// TIA Portal V20 export
FUNCTION "06 T4 LANT Output" : Void   // FC1612, LAD
TITLE = OUTPUT
{ S7_Optimized_Access := 'TRUE' }
// stored: AutoNumber false, SetENOAutomatically false
   VAR_TEMP
      Aux_real : Real;
      Aux_dint : DInt;
      Aux_uint : UInt;
      Aux_Bool : Bool;
      Aux_OS : Bool;
   END_VAR
   VAR_TEMP   // added for the SCL form of the ladder/FBD networks
      _w1 : Bool;
      _w2 : Bool;
      _w3 : Bool;
   END_VAR
BEGIN

REGION Network 1: ============= INTERLOCKS MOVING FORWARD LANT =============
END_REGION

REGION Network 2: Interlocks Move FORWARD LANT - Permanent Conditions
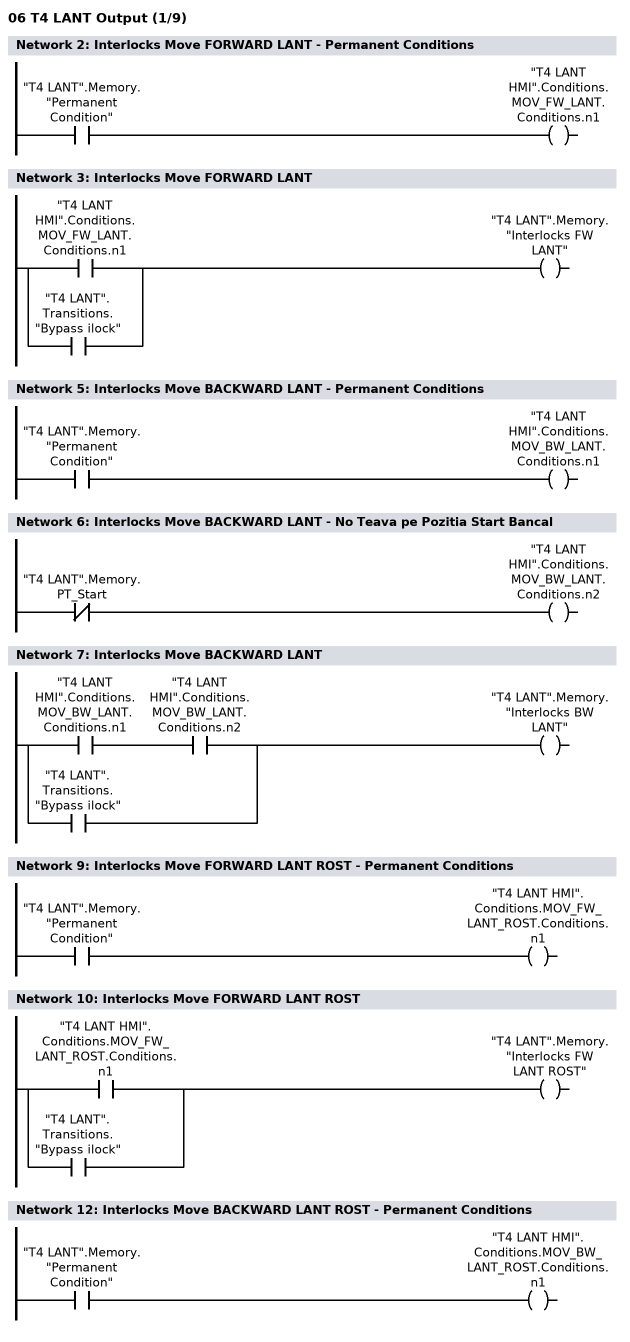
   RUNG wire#powerrail
      Contact( "T4 LANT".Memory."Permanent Condition" )
      Coil( "T4 LANT HMI".Conditions.MOV_FW_LANT.Conditions.n1 )
   END_RUNG
   // the same network as SCL:
   "T4 LANT HMI".Conditions.MOV_FW_LANT.Conditions.n1 := "T4 LANT".Memory."Permanent Condition";
END_REGION

REGION Network 3: Interlocks Move FORWARD LANT
   RUNG wire#powerrail
      Contact( "T4 LANT HMI".Conditions.MOV_FW_LANT.Conditions.n1 )
      wire#w1
      Coil( "T4 LANT".Memory."Interlocks FW LANT" )
   END_RUNG
   RUNG wire#powerrail
      Contact( "T4 LANT".Transitions."Bypass ilock" )
   END_RUNG wire#w1
   // the same network as SCL:
   "T4 LANT".Memory."Interlocks FW LANT" := "T4 LANT HMI".Conditions.MOV_FW_LANT.Conditions.n1 OR "T4 LANT".Transitions."Bypass ilock";
END_REGION

REGION Network 4: ============= INTERLOCKS MOVING BACKWARD LANT =============
END_REGION

REGION Network 5: Interlocks Move BACKWARD LANT - Permanent Conditions
   RUNG wire#powerrail
      Contact( "T4 LANT".Memory."Permanent Condition" )
      Coil( "T4 LANT HMI".Conditions.MOV_BW_LANT.Conditions.n1 )
   END_RUNG
   // the same network as SCL:
   "T4 LANT HMI".Conditions.MOV_BW_LANT.Conditions.n1 := "T4 LANT".Memory."Permanent Condition";
END_REGION

REGION Network 6: Interlocks Move BACKWARD LANT - No Teava pe Pozitia Start Bancal
   RUNG wire#powerrail
      I_Contact( "T4 LANT".Memory.PT_Start )
      Coil( "T4 LANT HMI".Conditions.MOV_BW_LANT.Conditions.n2 )
   END_RUNG
   // the same network as SCL:
   "T4 LANT HMI".Conditions.MOV_BW_LANT.Conditions.n2 := NOT "T4 LANT".Memory.PT_Start;
END_REGION

REGION Network 7: Interlocks Move BACKWARD LANT
   RUNG wire#powerrail
      Contact( "T4 LANT HMI".Conditions.MOV_BW_LANT.Conditions.n1 )
      Contact( "T4 LANT HMI".Conditions.MOV_BW_LANT.Conditions.n2 )
      wire#w1
      Coil( "T4 LANT".Memory."Interlocks BW LANT" )
   END_RUNG
   RUNG wire#powerrail
      Contact( "T4 LANT".Transitions."Bypass ilock" )
   END_RUNG wire#w1
   // the same network as SCL:
   "T4 LANT".Memory."Interlocks BW LANT" := ("T4 LANT HMI".Conditions.MOV_BW_LANT.Conditions.n1 AND "T4 LANT HMI".Conditions.MOV_BW_LANT.Conditions.n2) OR "T4 LANT".Transitions."Bypass ilock";
END_REGION

REGION Network 8: ============= INTERLOCKS MOVING FORWARD LANT ROST =============
END_REGION

REGION Network 9: Interlocks Move FORWARD LANT ROST - Permanent Conditions
   RUNG wire#powerrail
      Contact( "T4 LANT".Memory."Permanent Condition" )
      Coil( "T4 LANT HMI".Conditions.MOV_FW_LANT_ROST.Conditions.n1 )
   END_RUNG
   // the same network as SCL:
   "T4 LANT HMI".Conditions.MOV_FW_LANT_ROST.Conditions.n1 := "T4 LANT".Memory."Permanent Condition";
END_REGION

REGION Network 10: Interlocks Move FORWARD LANT ROST
   RUNG wire#powerrail
      Contact( "T4 LANT HMI".Conditions.MOV_FW_LANT_ROST.Conditions.n1 )
      wire#w1
      Coil( "T4 LANT".Memory."Interlocks FW LANT ROST" )
   END_RUNG
   RUNG wire#powerrail
      Contact( "T4 LANT".Transitions."Bypass ilock" )
   END_RUNG wire#w1
   // the same network as SCL:
   "T4 LANT".Memory."Interlocks FW LANT ROST" := "T4 LANT HMI".Conditions.MOV_FW_LANT_ROST.Conditions.n1 OR "T4 LANT".Transitions."Bypass ilock";
END_REGION

REGION Network 11: ============= INTERLOCKS MOVING BACKWARD LANT ROST =============
END_REGION

REGION Network 12: Interlocks Move BACKWARD LANT ROST - Permanent Conditions
   RUNG wire#powerrail
      Contact( "T4 LANT".Memory."Permanent Condition" )
      Coil( "T4 LANT HMI".Conditions.MOV_BW_LANT_ROST.Conditions.n1 )
   END_RUNG
   // the same network as SCL:
   "T4 LANT HMI".Conditions.MOV_BW_LANT_ROST.Conditions.n1 := "T4 LANT".Memory."Permanent Condition";
END_REGION

REGION Network 13: Interlocks Move BACKWARD LANT ROST - No TimeOut Cuplare/Decupl. Alim.Inv.LantRost
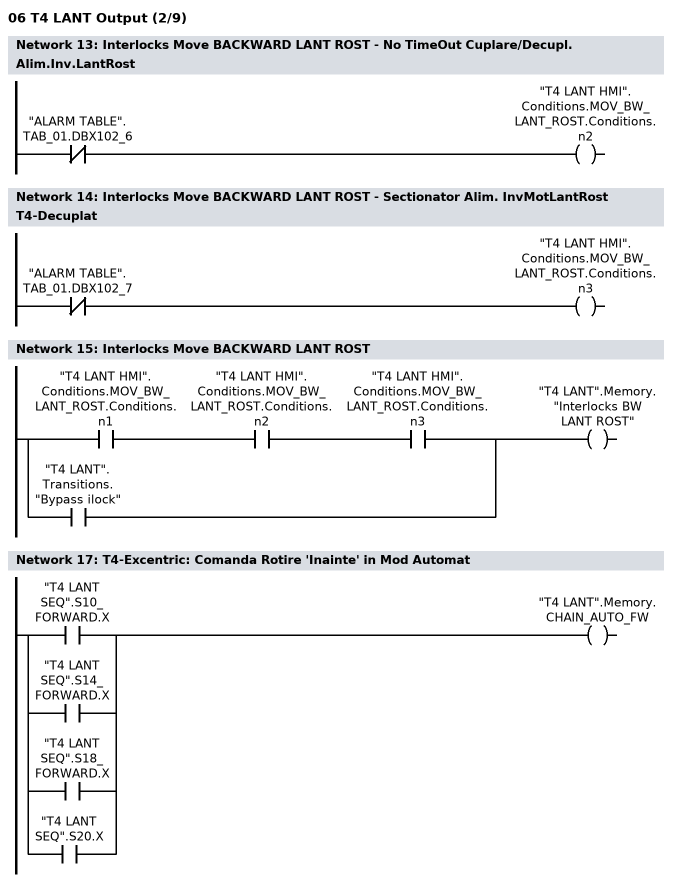
   RUNG wire#powerrail
      I_Contact( "ALARM TABLE".TAB_01.DBX102_6 )
      Coil( "T4 LANT HMI".Conditions.MOV_BW_LANT_ROST.Conditions.n2 )
   END_RUNG
   // the same network as SCL:
   "T4 LANT HMI".Conditions.MOV_BW_LANT_ROST.Conditions.n2 := NOT "ALARM TABLE".TAB_01.DBX102_6;
END_REGION

REGION Network 14: Interlocks Move BACKWARD LANT ROST - Sectionator Alim. InvMotLantRost T4-Decuplat
   RUNG wire#powerrail
      I_Contact( "ALARM TABLE".TAB_01.DBX102_7 )
      Coil( "T4 LANT HMI".Conditions.MOV_BW_LANT_ROST.Conditions.n3 )
   END_RUNG
   // the same network as SCL:
   "T4 LANT HMI".Conditions.MOV_BW_LANT_ROST.Conditions.n3 := NOT "ALARM TABLE".TAB_01.DBX102_7;
END_REGION

REGION Network 15: Interlocks Move BACKWARD LANT ROST
   RUNG wire#powerrail
      Contact( "T4 LANT HMI".Conditions.MOV_BW_LANT_ROST.Conditions.n1 )
      Contact( "T4 LANT HMI".Conditions.MOV_BW_LANT_ROST.Conditions.n2 )
      Contact( "T4 LANT HMI".Conditions.MOV_BW_LANT_ROST.Conditions.n3 )
      wire#w1
      Coil( "T4 LANT".Memory."Interlocks BW LANT ROST" )
   END_RUNG
   RUNG wire#powerrail
      Contact( "T4 LANT".Transitions."Bypass ilock" )
   END_RUNG wire#w1
   // the same network as SCL:
   "T4 LANT".Memory."Interlocks BW LANT ROST" := ("T4 LANT HMI".Conditions.MOV_BW_LANT_ROST.Conditions.n1 AND "T4 LANT HMI".Conditions.MOV_BW_LANT_ROST.Conditions.n2 AND "T4 LANT HMI".Conditions.MOV_BW_LANT_ROST.Conditions.n3) OR "T4 LANT".Transitions."Bypass ilock";
END_REGION

REGION Network 16: ============ COMMANDS ============
END_REGION

REGION Network 17: T4-Excentric: Comanda Rotire 'Inainte' in Mod Automat
   RUNG wire#powerrail
      Contact( "T4 LANT SEQ".S10_FORWARD.X )
      wire#w1
      Coil( "T4 LANT".Memory.CHAIN_AUTO_FW )
   END_RUNG
   RUNG wire#powerrail
      Contact( "T4 LANT SEQ".S14_FORWARD.X )
   END_RUNG wire#w1
   RUNG wire#powerrail
      Contact( "T4 LANT SEQ".S18_FORWARD.X )
   END_RUNG wire#w1
   RUNG wire#powerrail
      Contact( "T4 LANT SEQ".S20.X )
   END_RUNG wire#w1
   // the same network as SCL:
   "T4 LANT".Memory.CHAIN_AUTO_FW := "T4 LANT SEQ".S10_FORWARD.X OR "T4 LANT SEQ".S14_FORWARD.X OR "T4 LANT SEQ".S18_FORWARD.X OR "T4 LANT SEQ".S20.X;
END_REGION

REGION Network 18: T4-Lant: Deplasare 'Inainte'
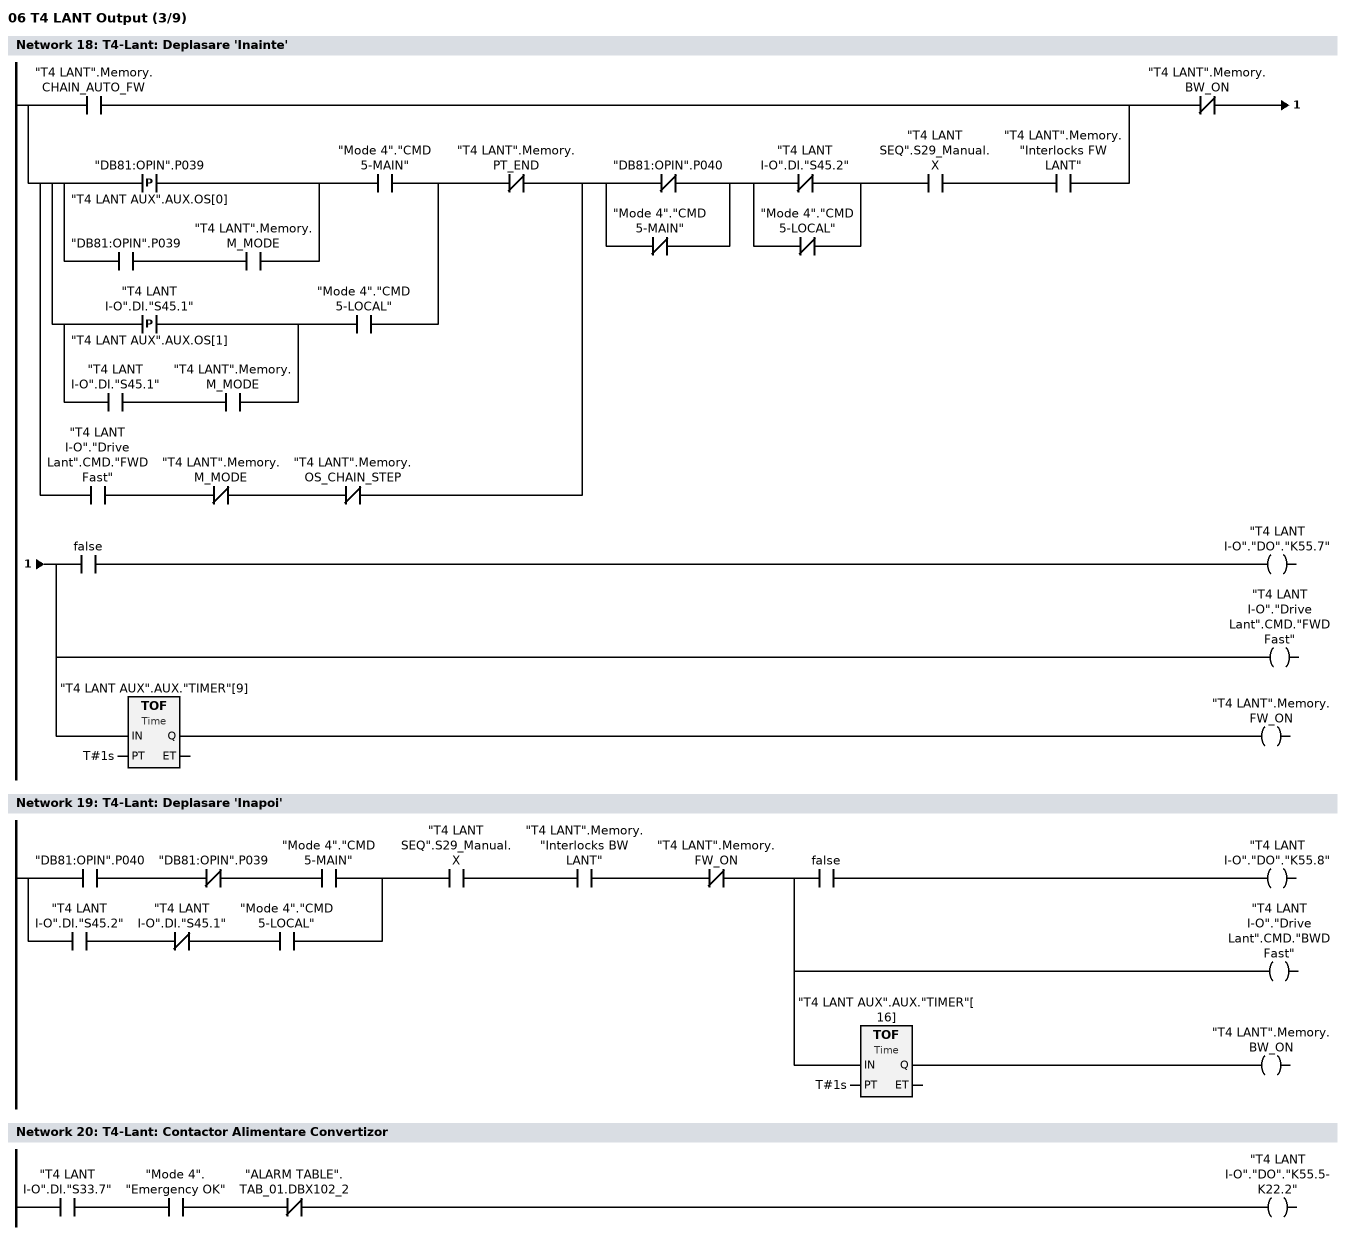
   RUNG wire#powerrail
      Contact( "T4 LANT".Memory.CHAIN_AUTO_FW )
      wire#w1
      I_Contact( "T4 LANT".Memory.BW_ON )
      wire#w8
      Contact( false )
      Coil( "T4 LANT I-O"."DO"."K55.7" )
   END_RUNG
   RUNG wire#powerrail
      P_Contact(operand := "DB81:OPIN".P039, bit := "T4 LANT AUX".AUX.OS[0])
      wire#w2
      Contact( "Mode 4"."CMD 5-MAIN" )
      wire#w3
      I_Contact( "T4 LANT".Memory.PT_END )
      wire#w5
      I_Contact( "DB81:OPIN".P040 )
      wire#w6
      I_Contact( "T4 LANT I-O".DI."S45.2" )
      wire#w7
      Contact( "T4 LANT SEQ".S29_Manual.X )
      Contact( "T4 LANT".Memory."Interlocks FW LANT" )
   END_RUNG wire#w1
   RUNG wire#powerrail
      Contact( "DB81:OPIN".P039 )
      Contact( "T4 LANT".Memory.M_MODE )
   END_RUNG wire#w2
   RUNG wire#powerrail
      P_Contact(operand := "T4 LANT I-O".DI."S45.1", bit := "T4 LANT AUX".AUX.OS[1])
      wire#w4
      Contact( "Mode 4"."CMD 5-LOCAL" )
   END_RUNG wire#w3
   RUNG wire#powerrail
      Contact( "T4 LANT I-O".DI."S45.1" )
      Contact( "T4 LANT".Memory.M_MODE )
   END_RUNG wire#w4
   RUNG wire#powerrail
      Contact( "T4 LANT I-O"."Drive Lant".CMD."FWD Fast" )
      I_Contact( "T4 LANT".Memory.M_MODE )
      I_Contact( "T4 LANT".Memory.OS_CHAIN_STEP )
   END_RUNG wire#w5
   RUNG wire#w5
      I_Contact( "Mode 4"."CMD 5-MAIN" )
   END_RUNG wire#w6
   RUNG wire#w6
      I_Contact( "Mode 4"."CMD 5-LOCAL" )
   END_RUNG wire#w7
   RUNG wire#w8
      Coil( "T4 LANT I-O"."Drive Lant".CMD."FWD Fast" )
   END_RUNG
   RUNG wire#w8
      { S7_Templates := "time_type := Time" } "T4 LANT AUX".AUX."TIMER"[9].TOF(pt := T#1s, et =>)
      Coil( "T4 LANT".Memory.FW_ON )
   END_RUNG
   // the same network as SCL:
   #_w1 := "DB81:OPIN".P039 AND NOT "T4 LANT AUX".AUX.OS[0];   // rising edge of "DB81:OPIN".P039
   "T4 LANT AUX".AUX.OS[0] := "DB81:OPIN".P039;
   #_w2 := "T4 LANT I-O".DI."S45.1" AND NOT "T4 LANT AUX".AUX.OS[1];   // rising edge of "T4 LANT I-O".DI."S45.1"
   "T4 LANT AUX".AUX.OS[1] := "T4 LANT I-O".DI."S45.1";
   #_w3 := ("T4 LANT".Memory.CHAIN_AUTO_FW OR ((((((#_w1 OR ("DB81:OPIN".P039 AND "T4 LANT".Memory.M_MODE)) AND "Mode 4"."CMD 5-MAIN") OR ((#_w2 OR ("T4 LANT I-O".DI."S45.1" AND "T4 LANT".Memory.M_MODE)) AND "Mode 4"."CMD 5-LOCAL")) AND NOT "T4 LANT".Memory.PT_END) OR ("T4 LANT I-O"."Drive Lant".CMD."FWD Fast" AND NOT "T4 LANT".Memory.M_MODE AND NOT "T4 LANT".Memory.OS_CHAIN_STEP)) AND (NOT "DB81:OPIN".P040 OR NOT "Mode 4"."CMD 5-MAIN") AND (NOT "T4 LANT I-O".DI."S45.2" OR NOT "Mode 4"."CMD 5-LOCAL") AND "T4 LANT SEQ".S29_Manual.X AND "T4 LANT".Memory."Interlocks FW LANT")) AND NOT "T4 LANT".Memory.BW_ON;
   "T4 LANT I-O"."DO"."K55.7" := #_w3 AND false;
   "T4 LANT I-O"."Drive Lant".CMD."FWD Fast" := #_w3;
   "T4 LANT AUX".AUX."TIMER"[9].TOF(IN := #_w3, PT := T#1s);
   "T4 LANT".Memory.FW_ON := "T4 LANT AUX".AUX."TIMER"[9].Q;
END_REGION

REGION Network 19: T4-Lant: Deplasare 'Inapoi'
   RUNG wire#powerrail
      Contact( "DB81:OPIN".P040 )
      I_Contact( "DB81:OPIN".P039 )
      Contact( "Mode 4"."CMD 5-MAIN" )
      wire#w1
      Contact( "T4 LANT SEQ".S29_Manual.X )
      Contact( "T4 LANT".Memory."Interlocks BW LANT" )
      I_Contact( "T4 LANT".Memory.FW_ON )
      wire#w2
      Contact( false )
      Coil( "T4 LANT I-O"."DO"."K55.8" )
   END_RUNG
   RUNG wire#powerrail
      Contact( "T4 LANT I-O".DI."S45.2" )
      I_Contact( "T4 LANT I-O".DI."S45.1" )
      Contact( "Mode 4"."CMD 5-LOCAL" )
   END_RUNG wire#w1
   RUNG wire#w2
      Coil( "T4 LANT I-O"."Drive Lant".CMD."BWD Fast" )
   END_RUNG
   RUNG wire#w2
      { S7_Templates := "time_type := Time" } "T4 LANT AUX".AUX."TIMER"[16].TOF(pt := T#1s, et =>)
      Coil( "T4 LANT".Memory.BW_ON )
   END_RUNG
   // the same network as SCL:
   #_w1 := (("DB81:OPIN".P040 AND NOT "DB81:OPIN".P039 AND "Mode 4"."CMD 5-MAIN") OR ("T4 LANT I-O".DI."S45.2" AND NOT "T4 LANT I-O".DI."S45.1" AND "Mode 4"."CMD 5-LOCAL")) AND "T4 LANT SEQ".S29_Manual.X AND "T4 LANT".Memory."Interlocks BW LANT" AND NOT "T4 LANT".Memory.FW_ON;
   "T4 LANT I-O"."DO"."K55.8" := #_w1 AND false;
   "T4 LANT I-O"."Drive Lant".CMD."BWD Fast" := #_w1;
   "T4 LANT AUX".AUX."TIMER"[16].TOF(IN := #_w1, PT := T#1s);
   "T4 LANT".Memory.BW_ON := "T4 LANT AUX".AUX."TIMER"[16].Q;
END_REGION

REGION Network 20: T4-Lant: Contactor Alimentare Convertizor
   RUNG wire#powerrail
      Contact( "T4 LANT I-O".DI."S33.7" )
      Contact( "Mode 4"."Emergency OK" )
      I_Contact( "ALARM TABLE".TAB_01.DBX102_2 )
      Coil( "T4 LANT I-O"."DO"."K55.5-K22.2" )
   END_RUNG
   // the same network as SCL:
   "T4 LANT I-O"."DO"."K55.5-K22.2" := "T4 LANT I-O".DI."S33.7" AND "Mode 4"."Emergency OK" AND NOT "ALARM TABLE".TAB_01.DBX102_2;
END_REGION

REGION Network 21: T4-LantRost: Comanda Deplasare 'Inainte'
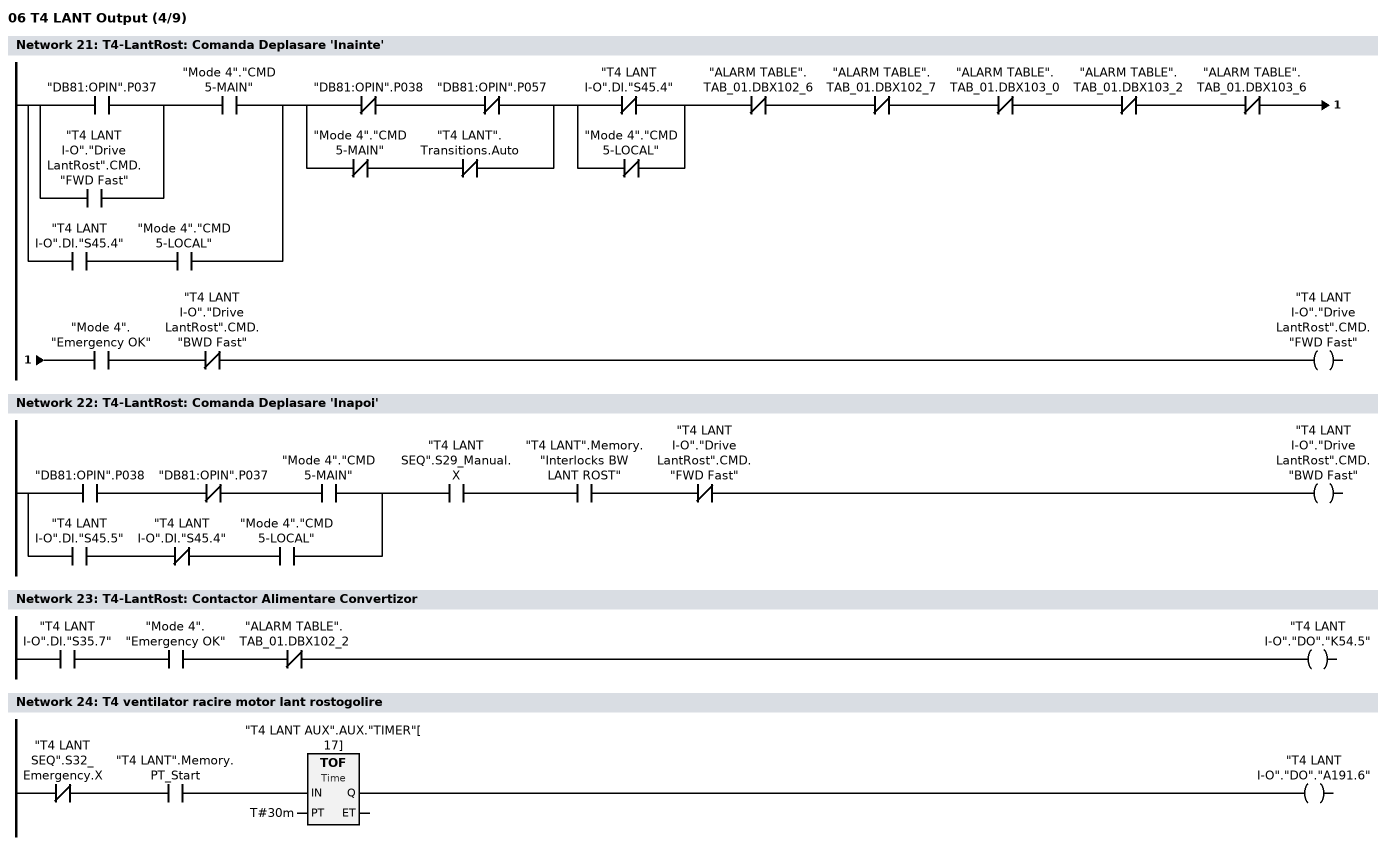
   RUNG wire#powerrail
      Contact( "DB81:OPIN".P037 )
      wire#w1
      Contact( "Mode 4"."CMD 5-MAIN" )
      wire#w2
      I_Contact( "DB81:OPIN".P038 )
      I_Contact( "DB81:OPIN".P057 )
      wire#w3
      I_Contact( "T4 LANT I-O".DI."S45.4" )
      wire#w4
      I_Contact( "ALARM TABLE".TAB_01.DBX102_6 )
      I_Contact( "ALARM TABLE".TAB_01.DBX102_7 )
      I_Contact( "ALARM TABLE".TAB_01.DBX103_0 )
      I_Contact( "ALARM TABLE".TAB_01.DBX103_2 )
      I_Contact( "ALARM TABLE".TAB_01.DBX103_6 )
      Contact( "Mode 4"."Emergency OK" )
      I_Contact( "T4 LANT I-O"."Drive LantRost".CMD."BWD Fast" )
      Coil( "T4 LANT I-O"."Drive LantRost".CMD."FWD Fast" )
   END_RUNG
   RUNG wire#powerrail
      Contact( "T4 LANT I-O"."Drive LantRost".CMD."FWD Fast" )
   END_RUNG wire#w1
   RUNG wire#powerrail
      Contact( "T4 LANT I-O".DI."S45.4" )
      Contact( "Mode 4"."CMD 5-LOCAL" )
   END_RUNG wire#w2
   RUNG wire#w2
      I_Contact( "Mode 4"."CMD 5-MAIN" )
      I_Contact( "T4 LANT".Transitions.Auto )
   END_RUNG wire#w3
   RUNG wire#w3
      I_Contact( "Mode 4"."CMD 5-LOCAL" )
   END_RUNG wire#w4
   // the same network as SCL:
   "T4 LANT I-O"."Drive LantRost".CMD."FWD Fast" := ((("DB81:OPIN".P037 OR "T4 LANT I-O"."Drive LantRost".CMD."FWD Fast") AND "Mode 4"."CMD 5-MAIN") OR ("T4 LANT I-O".DI."S45.4" AND "Mode 4"."CMD 5-LOCAL")) AND ((NOT "DB81:OPIN".P038 AND NOT "DB81:OPIN".P057) OR (NOT "Mode 4"."CMD 5-MAIN" AND NOT "T4 LANT".Transitions.Auto)) AND (NOT "T4 LANT I-O".DI."S45.4" OR NOT "Mode 4"."CMD 5-LOCAL") AND NOT "ALARM TABLE".TAB_01.DBX102_6 AND NOT "ALARM TABLE".TAB_01.DBX102_7 AND NOT "ALARM TABLE".TAB_01.DBX103_0 AND NOT "ALARM TABLE".TAB_01.DBX103_2 AND NOT "ALARM TABLE".TAB_01.DBX103_6 AND "Mode 4"."Emergency OK" AND NOT "T4 LANT I-O"."Drive LantRost".CMD."BWD Fast";
END_REGION

REGION Network 22: T4-LantRost: Comanda Deplasare 'Inapoi'
   RUNG wire#powerrail
      Contact( "DB81:OPIN".P038 )
      I_Contact( "DB81:OPIN".P037 )
      Contact( "Mode 4"."CMD 5-MAIN" )
      wire#w1
      Contact( "T4 LANT SEQ".S29_Manual.X )
      Contact( "T4 LANT".Memory."Interlocks BW LANT ROST" )
      I_Contact( "T4 LANT I-O"."Drive LantRost".CMD."FWD Fast" )
      Coil( "T4 LANT I-O"."Drive LantRost".CMD."BWD Fast" )
   END_RUNG
   RUNG wire#powerrail
      Contact( "T4 LANT I-O".DI."S45.5" )
      I_Contact( "T4 LANT I-O".DI."S45.4" )
      Contact( "Mode 4"."CMD 5-LOCAL" )
   END_RUNG wire#w1
   // the same network as SCL:
   "T4 LANT I-O"."Drive LantRost".CMD."BWD Fast" := (("DB81:OPIN".P038 AND NOT "DB81:OPIN".P037 AND "Mode 4"."CMD 5-MAIN") OR ("T4 LANT I-O".DI."S45.5" AND NOT "T4 LANT I-O".DI."S45.4" AND "Mode 4"."CMD 5-LOCAL")) AND "T4 LANT SEQ".S29_Manual.X AND "T4 LANT".Memory."Interlocks BW LANT ROST" AND NOT "T4 LANT I-O"."Drive LantRost".CMD."FWD Fast";
END_REGION

REGION Network 23: T4-LantRost: Contactor Alimentare Convertizor
   RUNG wire#powerrail
      Contact( "T4 LANT I-O".DI."S35.7" )
      Contact( "Mode 4"."Emergency OK" )
      I_Contact( "ALARM TABLE".TAB_01.DBX102_2 )
      Coil( "T4 LANT I-O"."DO"."K54.5" )
   END_RUNG
   // the same network as SCL:
   "T4 LANT I-O"."DO"."K54.5" := "T4 LANT I-O".DI."S35.7" AND "Mode 4"."Emergency OK" AND NOT "ALARM TABLE".TAB_01.DBX102_2;
END_REGION

REGION Network 24: T4 ventilator racire motor lant rostogolire
   RUNG wire#powerrail
      I_Contact( "T4 LANT SEQ".S32_Emergency.X )
      Contact( "T4 LANT".Memory.PT_Start )
      { S7_Templates := "time_type := Time" } "T4 LANT AUX".AUX."TIMER"[17].TOF(pt := T#30m, et =>)
      Coil( "T4 LANT I-O"."DO"."A191.6" )
   END_RUNG
   // the same network as SCL:
   "T4 LANT AUX".AUX."TIMER"[17].TOF(IN := NOT "T4 LANT SEQ".S32_Emergency.X AND "T4 LANT".Memory.PT_Start,
                           PT := T#30m);
   "T4 LANT I-O"."DO"."A191.6" := "T4 LANT AUX".AUX."TIMER"[17].Q;
END_REGION

REGION Network 25: T4-Lant: Ciclu Rapid: Viteza Referinta Incarcare
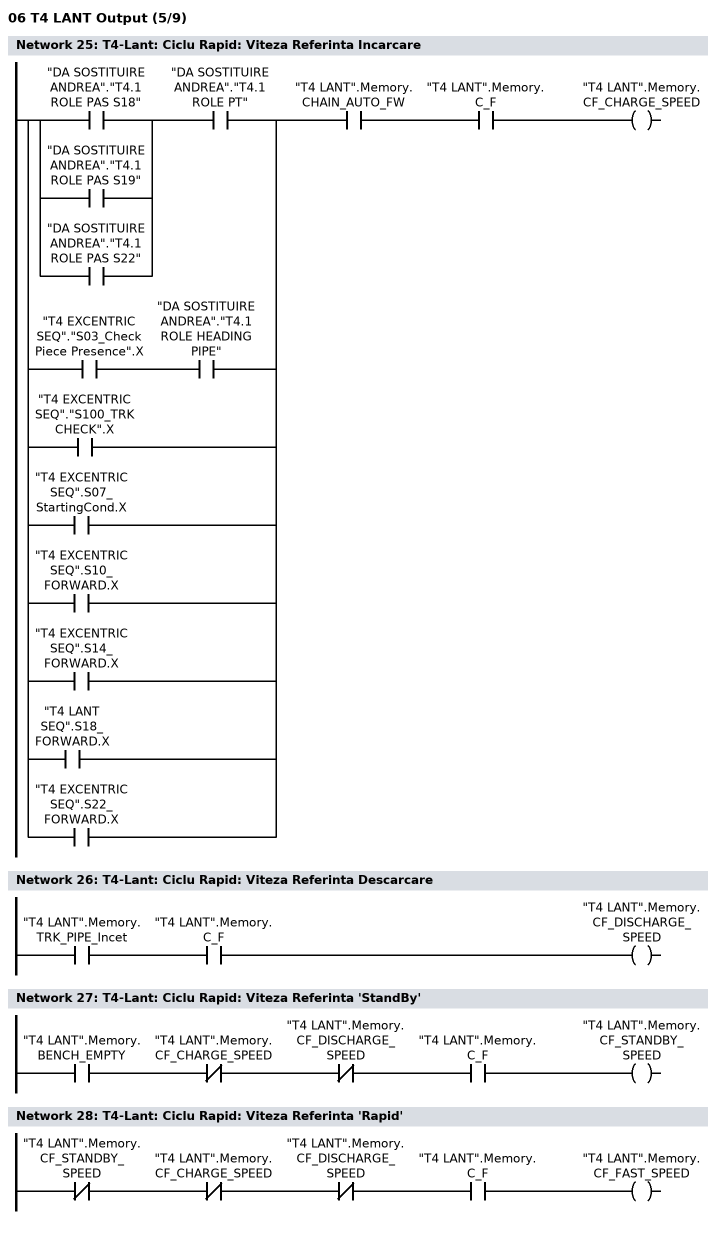
   RUNG wire#powerrail
      Contact( "DA SOSTITUIRE ANDREA"."T4.1 ROLE PAS S18" )
      wire#w1
      Contact( "DA SOSTITUIRE ANDREA"."T4.1 ROLE PT" )
      wire#w2
      Contact( "T4 LANT".Memory.CHAIN_AUTO_FW )
      Contact( "T4 LANT".Memory.C_F )
      Coil( "T4 LANT".Memory.CF_CHARGE_SPEED )
   END_RUNG
   RUNG wire#powerrail
      Contact( "DA SOSTITUIRE ANDREA"."T4.1 ROLE PAS S19" )
   END_RUNG wire#w1
   RUNG wire#powerrail
      Contact( "DA SOSTITUIRE ANDREA"."T4.1 ROLE PAS S22" )
   END_RUNG wire#w1
   RUNG wire#powerrail
      Contact( "T4 EXCENTRIC SEQ"."S03_Check Piece Presence".X )
      Contact( "DA SOSTITUIRE ANDREA"."T4.1 ROLE HEADING PIPE" )
   END_RUNG wire#w2
   RUNG wire#powerrail
      Contact( "T4 EXCENTRIC SEQ"."S100_TRK CHECK".X )
   END_RUNG wire#w2
   RUNG wire#powerrail
      Contact( "T4 EXCENTRIC SEQ".S07_StartingCond.X )
   END_RUNG wire#w2
   RUNG wire#powerrail
      Contact( "T4 EXCENTRIC SEQ".S10_FORWARD.X )
   END_RUNG wire#w2
   RUNG wire#powerrail
      Contact( "T4 EXCENTRIC SEQ".S14_FORWARD.X )
   END_RUNG wire#w2
   RUNG wire#powerrail
      Contact( "T4 LANT SEQ".S18_FORWARD.X )
   END_RUNG wire#w2
   RUNG wire#powerrail
      Contact( "T4 EXCENTRIC SEQ".S22_FORWARD.X )
   END_RUNG wire#w2
   // the same network as SCL:
   "T4 LANT".Memory.CF_CHARGE_SPEED := ((("DA SOSTITUIRE ANDREA"."T4.1 ROLE PAS S18" OR "DA SOSTITUIRE ANDREA"."T4.1 ROLE PAS S19" OR "DA SOSTITUIRE ANDREA"."T4.1 ROLE PAS S22") AND "DA SOSTITUIRE ANDREA"."T4.1 ROLE PT") OR ("T4 EXCENTRIC SEQ"."S03_Check Piece Presence".X AND "DA SOSTITUIRE ANDREA"."T4.1 ROLE HEADING PIPE") OR "T4 EXCENTRIC SEQ"."S100_TRK CHECK".X OR "T4 EXCENTRIC SEQ".S07_StartingCond.X OR "T4 EXCENTRIC SEQ".S10_FORWARD.X OR "T4 EXCENTRIC SEQ".S14_FORWARD.X OR "T4 LANT SEQ".S18_FORWARD.X OR "T4 EXCENTRIC SEQ".S22_FORWARD.X) AND "T4 LANT".Memory.CHAIN_AUTO_FW AND "T4 LANT".Memory.C_F;
END_REGION

REGION Network 26: T4-Lant: Ciclu Rapid: Viteza Referinta Descarcare
   RUNG wire#powerrail
      Contact( "T4 LANT".Memory.TRK_PIPE_Incet )
      Contact( "T4 LANT".Memory.C_F )
      Coil( "T4 LANT".Memory.CF_DISCHARGE_SPEED )
   END_RUNG
   // the same network as SCL:
   "T4 LANT".Memory.CF_DISCHARGE_SPEED := "T4 LANT".Memory.TRK_PIPE_Incet AND "T4 LANT".Memory.C_F;
END_REGION

REGION Network 27: T4-Lant: Ciclu Rapid: Viteza Referinta 'StandBy'
   RUNG wire#powerrail
      Contact( "T4 LANT".Memory.BENCH_EMPTY )
      I_Contact( "T4 LANT".Memory.CF_CHARGE_SPEED )
      I_Contact( "T4 LANT".Memory.CF_DISCHARGE_SPEED )
      Contact( "T4 LANT".Memory.C_F )
      Coil( "T4 LANT".Memory.CF_STANDBY_SPEED )
   END_RUNG
   // the same network as SCL:
   "T4 LANT".Memory.CF_STANDBY_SPEED := "T4 LANT".Memory.BENCH_EMPTY AND NOT "T4 LANT".Memory.CF_CHARGE_SPEED AND NOT "T4 LANT".Memory.CF_DISCHARGE_SPEED AND "T4 LANT".Memory.C_F;
END_REGION

REGION Network 28: T4-Lant: Ciclu Rapid: Viteza Referinta 'Rapid'
   RUNG wire#powerrail
      I_Contact( "T4 LANT".Memory.CF_STANDBY_SPEED )
      I_Contact( "T4 LANT".Memory.CF_CHARGE_SPEED )
      I_Contact( "T4 LANT".Memory.CF_DISCHARGE_SPEED )
      Contact( "T4 LANT".Memory.C_F )
      Coil( "T4 LANT".Memory.CF_FAST_SPEED )
   END_RUNG
   // the same network as SCL:
   "T4 LANT".Memory.CF_FAST_SPEED := NOT "T4 LANT".Memory.CF_STANDBY_SPEED AND NOT "T4 LANT".Memory.CF_CHARGE_SPEED AND NOT "T4 LANT".Memory.CF_DISCHARGE_SPEED AND "T4 LANT".Memory.C_F;
END_REGION

REGION Network 29: T4-Lant: Viteza Teava 'Inainte' in Mod Automat [m/min *10]
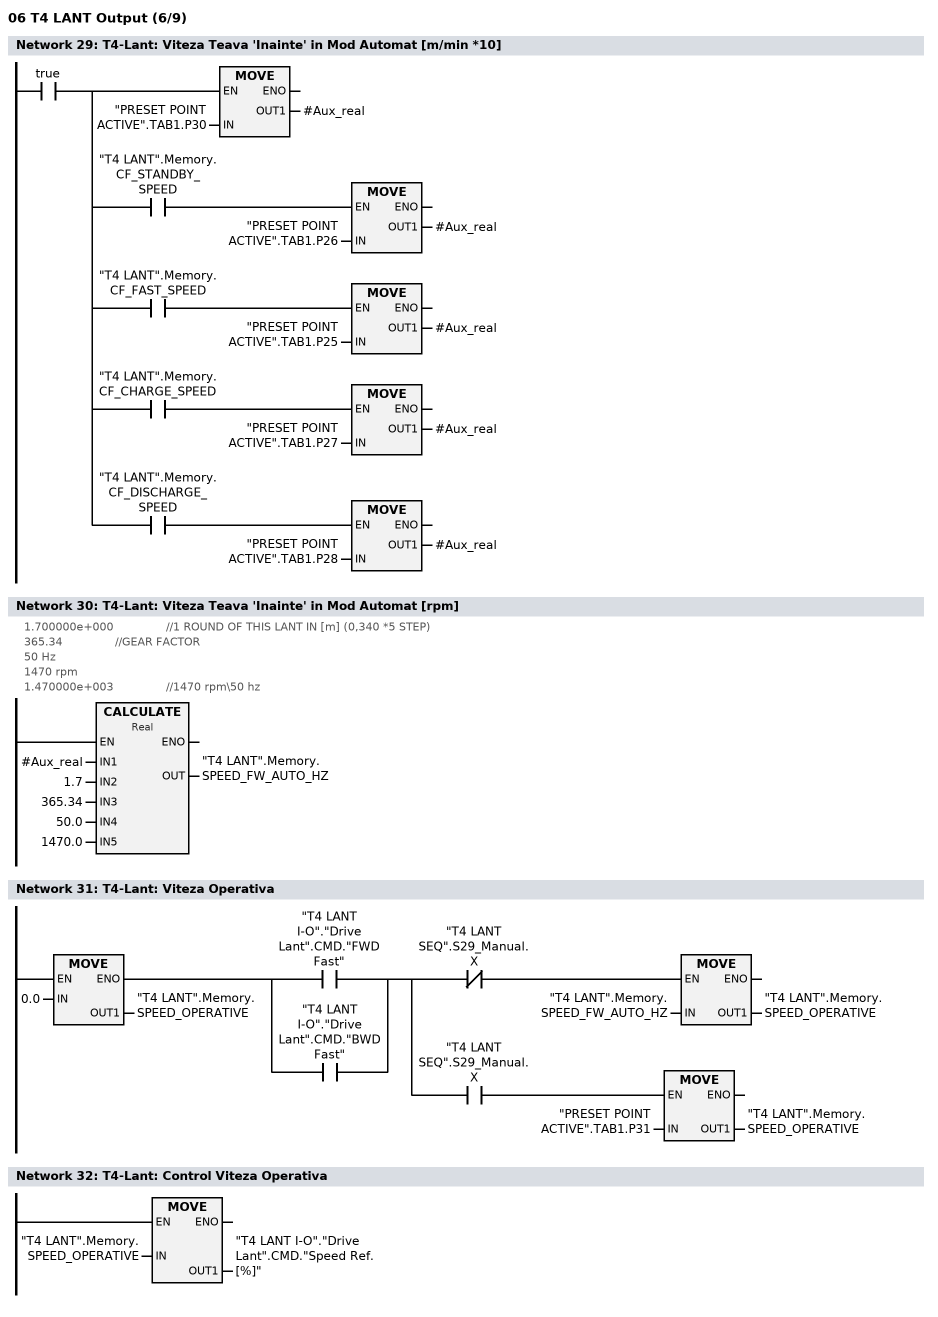
   RUNG wire#powerrail
      Contact( true )
      wire#w1
      Move(in := "PRESET POINT ACTIVE".TAB1.P30, out1 => #Aux_real)
   END_RUNG
   RUNG wire#w1
      Contact( "T4 LANT".Memory.CF_STANDBY_SPEED )
      Move(in := "PRESET POINT ACTIVE".TAB1.P26, out1 => #Aux_real)
   END_RUNG
   RUNG wire#w1
      Contact( "T4 LANT".Memory.CF_FAST_SPEED )
      Move(in := "PRESET POINT ACTIVE".TAB1.P25, out1 => #Aux_real)
   END_RUNG
   RUNG wire#w1
      Contact( "T4 LANT".Memory.CF_CHARGE_SPEED )
      Move(in := "PRESET POINT ACTIVE".TAB1.P27, out1 => #Aux_real)
   END_RUNG
   RUNG wire#w1
      Contact( "T4 LANT".Memory.CF_DISCHARGE_SPEED )
      Move(in := "PRESET POINT ACTIVE".TAB1.P28, out1 => #Aux_real)
   END_RUNG
   // the same network as SCL:
   IF true THEN #Aux_real := "PRESET POINT ACTIVE".TAB1.P30; END_IF;
   IF true AND "T4 LANT".Memory.CF_STANDBY_SPEED THEN #Aux_real := "PRESET POINT ACTIVE".TAB1.P26; END_IF;
   IF true AND "T4 LANT".Memory.CF_FAST_SPEED THEN #Aux_real := "PRESET POINT ACTIVE".TAB1.P25; END_IF;
   IF true AND "T4 LANT".Memory.CF_CHARGE_SPEED THEN #Aux_real := "PRESET POINT ACTIVE".TAB1.P27; END_IF;
   IF true AND "T4 LANT".Memory.CF_DISCHARGE_SPEED THEN #Aux_real := "PRESET POINT ACTIVE".TAB1.P28; END_IF;
END_REGION

REGION Network 30: T4-Lant: Viteza Teava 'Inainte' in Mod Automat [rpm]
   // 1.700000e+000               //1 ROUND OF THIS LANT IN [m] (0,340 *5 STEP) 
   //  365.34               //GEAR FACTOR
   // 50 Hz
   // 1470 rpm
   // 1.470000e+003               //1470 rpm\50 hz
   RUNG wire#powerrail
      { S7_Templates := "SrcType := Real"; S7_Expression := "IN1/IN2*IN3*IN4/IN5" } Calculate(in1 := #Aux_real, in2 := 1.7, in3 := 365.34, in4 := 50.0, in5 := 1470.0, out => "T4 LANT".Memory.SPEED_FW_AUTO_HZ)
   END_RUNG
   // the same network as SCL:
   "T4 LANT".Memory.SPEED_FW_AUTO_HZ := #Aux_real/1.7*365.34*50.0/1470.0;
END_REGION

REGION Network 31: T4-Lant: Viteza Operativa
   RUNG wire#powerrail
      Move(in := 0.0, out1 => "T4 LANT".Memory.SPEED_OPERATIVE)
      wire#w1
      Contact( "T4 LANT I-O"."Drive Lant".CMD."FWD Fast" )
      wire#w2
      I_Contact( "T4 LANT SEQ".S29_Manual.X )
      Move(in := "T4 LANT".Memory.SPEED_FW_AUTO_HZ, out1 => "T4 LANT".Memory.SPEED_OPERATIVE)
   END_RUNG
   RUNG wire#w1
      Contact( "T4 LANT I-O"."Drive Lant".CMD."BWD Fast" )
   END_RUNG wire#w2
   RUNG wire#w2
      Contact( "T4 LANT SEQ".S29_Manual.X )
      Move(in := "PRESET POINT ACTIVE".TAB1.P31, out1 => "T4 LANT".Memory.SPEED_OPERATIVE)
   END_RUNG
   // the same network as SCL:
   "T4 LANT".Memory.SPEED_OPERATIVE := 0.0;
   #_w1 := "T4 LANT I-O"."Drive Lant".CMD."FWD Fast" OR "T4 LANT I-O"."Drive Lant".CMD."BWD Fast";
   IF #_w1 AND NOT "T4 LANT SEQ".S29_Manual.X THEN
       "T4 LANT".Memory.SPEED_OPERATIVE := "T4 LANT".Memory.SPEED_FW_AUTO_HZ;
   END_IF;
   IF #_w1 AND "T4 LANT SEQ".S29_Manual.X THEN
       "T4 LANT".Memory.SPEED_OPERATIVE := "PRESET POINT ACTIVE".TAB1.P31;
   END_IF;
END_REGION

REGION Network 32: T4-Lant: Control Viteza Operativa
   RUNG wire#powerrail
      Move(in := "T4 LANT".Memory.SPEED_OPERATIVE, out1 => "T4 LANT I-O"."Drive Lant".CMD."Speed Ref. [%]")
   END_RUNG
   // the same network as SCL:
   "T4 LANT I-O"."Drive Lant".CMD."Speed Ref. [%]" := "T4 LANT".Memory.SPEED_OPERATIVE;
END_REGION

REGION Network 33: T4-Lant: Contactor Frana
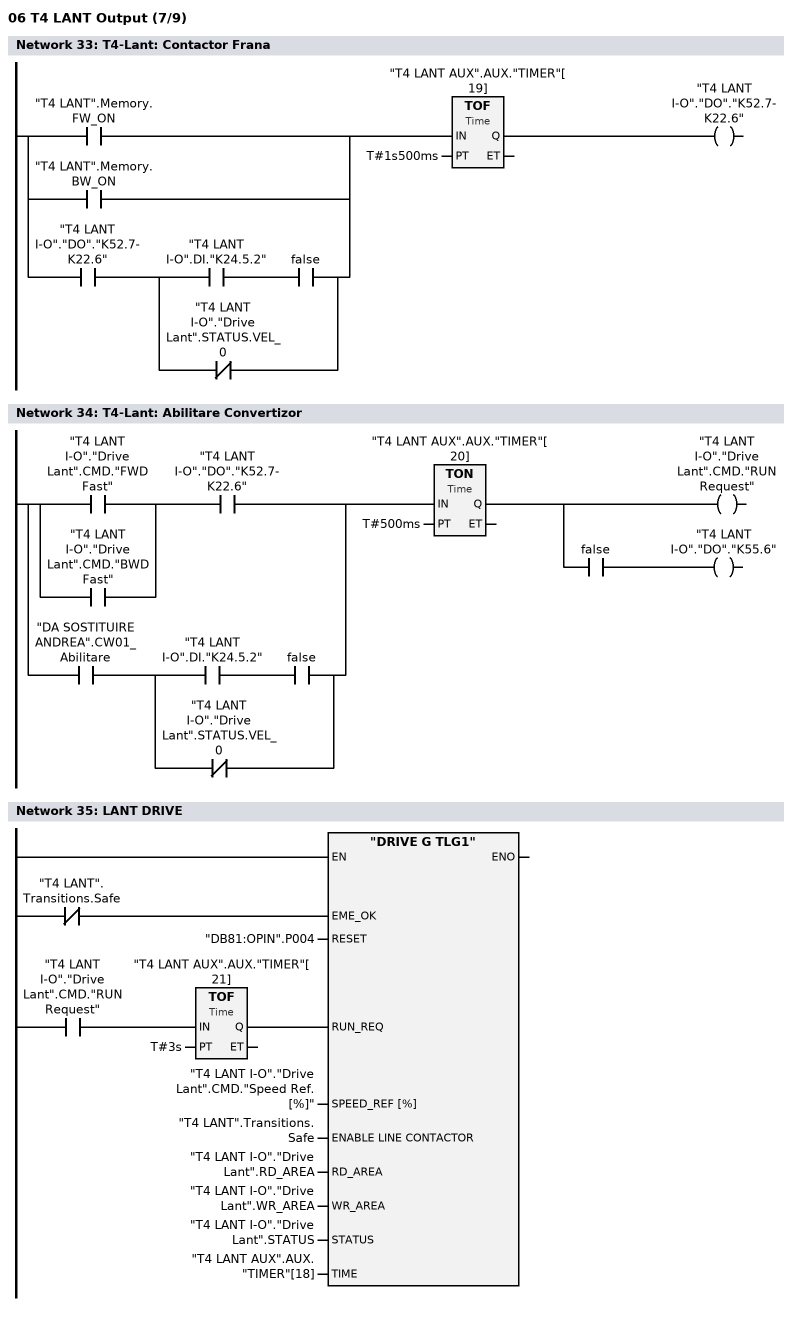
   RUNG wire#powerrail
      Contact( "T4 LANT".Memory.FW_ON )
      wire#w1
      { S7_Templates := "time_type := Time" } "T4 LANT AUX".AUX."TIMER"[19].TOF(pt := T#1s500ms, et =>)
      Coil( "T4 LANT I-O"."DO"."K52.7-K22.6" )
   END_RUNG
   RUNG wire#powerrail
      Contact( "T4 LANT".Memory.BW_ON )
   END_RUNG wire#w1
   RUNG wire#powerrail
      Contact( "T4 LANT I-O"."DO"."K52.7-K22.6" )
      wire#w2
      Contact( "T4 LANT I-O".DI."K24.5.2" )
      Contact( false )
   END_RUNG wire#w1
   RUNG wire#w2
      I_Contact( "T4 LANT I-O"."Drive Lant".STATUS.VEL_0 )
   END_RUNG wire#w1
   // the same network as SCL:
   "T4 LANT AUX".AUX."TIMER"[19].TOF(IN := "T4 LANT".Memory.FW_ON OR "T4 LANT".Memory.BW_ON OR ("T4 LANT I-O"."DO"."K52.7-K22.6" AND (("T4 LANT I-O".DI."K24.5.2" AND false) OR NOT "T4 LANT I-O"."Drive Lant".STATUS.VEL_0)),
                           PT := T#1s500ms);
   "T4 LANT I-O"."DO"."K52.7-K22.6" := "T4 LANT AUX".AUX."TIMER"[19].Q;
END_REGION

REGION Network 34: T4-Lant: Abilitare Convertizor
   RUNG wire#powerrail
      Contact( "T4 LANT I-O"."Drive Lant".CMD."FWD Fast" )
      wire#w1
      Contact( "T4 LANT I-O"."DO"."K52.7-K22.6" )
      wire#w2
      { S7_Templates := "time_type := Time" } "T4 LANT AUX".AUX."TIMER"[20].TON(pt := T#500ms, et =>)
      wire#w4
      Coil( "T4 LANT I-O"."Drive Lant".CMD."RUN Request" )
   END_RUNG
   RUNG wire#powerrail
      Contact( "T4 LANT I-O"."Drive Lant".CMD."BWD Fast" )
   END_RUNG wire#w1
   RUNG wire#powerrail
      Contact( "DA SOSTITUIRE ANDREA".CW01_Abilitare )
      wire#w3
      Contact( "T4 LANT I-O".DI."K24.5.2" )
      Contact( false )
   END_RUNG wire#w2
   RUNG wire#w3
      I_Contact( "T4 LANT I-O"."Drive Lant".STATUS.VEL_0 )
   END_RUNG wire#w2
   RUNG wire#w4
      Contact( false )
      Coil( "T4 LANT I-O"."DO"."K55.6" )
   END_RUNG
   // the same network as SCL:
   "T4 LANT AUX".AUX."TIMER"[20].TON(IN := (("T4 LANT I-O"."Drive Lant".CMD."FWD Fast" OR "T4 LANT I-O"."Drive Lant".CMD."BWD Fast") AND "T4 LANT I-O"."DO"."K52.7-K22.6") OR ("DA SOSTITUIRE ANDREA".CW01_Abilitare AND (("T4 LANT I-O".DI."K24.5.2" AND false) OR NOT "T4 LANT I-O"."Drive Lant".STATUS.VEL_0)),
                           PT := T#500ms);
   "T4 LANT I-O"."Drive Lant".CMD."RUN Request" := "T4 LANT AUX".AUX."TIMER"[20].Q;
   "T4 LANT I-O"."DO"."K55.6" := "T4 LANT AUX".AUX."TIMER"[20].Q AND false;
END_REGION

REGION Network 35: LANT DRIVE
   RUNG wire#powerrail
      "DRIVE G TLG1"(EME_OK := wire#w1, RUN_REQ := wire#w2, RESET := "DB81:OPIN".P004, "SPEED_REF [%]" := "T4 LANT I-O"."Drive Lant".CMD."Speed Ref. [%]", "ENABLE LINE CONTACTOR" := "T4 LANT".Transitions.Safe, RD_AREA := "T4 LANT I-O"."Drive Lant".RD_AREA, WR_AREA := "T4 LANT I-O"."Drive Lant".WR_AREA, STATUS := "T4 LANT I-O"."Drive Lant".STATUS, "TIME" := "T4 LANT AUX".AUX."TIMER"[18])
   END_RUNG
   RUNG wire#powerrail
      I_Contact( "T4 LANT".Transitions.Safe )
   END_RUNG wire#w1
   RUNG wire#powerrail
      Contact( "T4 LANT I-O"."Drive Lant".CMD."RUN Request" )
      { S7_Templates := "time_type := Time" } "T4 LANT AUX".AUX."TIMER"[21].TOF(pt := T#3s, et =>)
   END_RUNG wire#w2
   // the same network as SCL:
   "T4 LANT AUX".AUX."TIMER"[21].TOF(IN := "T4 LANT I-O"."Drive Lant".CMD."RUN Request", PT := T#3s);
   "DRIVE G TLG1"(EME_OK := NOT "T4 LANT".Transitions.Safe,
                  RESET := "DB81:OPIN".P004,
                  RUN_REQ := "T4 LANT AUX".AUX."TIMER"[21].Q,
                  "SPEED_REF [%]" := "T4 LANT I-O"."Drive Lant".CMD."Speed Ref. [%]",
                  "ENABLE LINE CONTACTOR" := "T4 LANT".Transitions.Safe,
                  RD_AREA := "T4 LANT I-O"."Drive Lant".RD_AREA,
                  WR_AREA := "T4 LANT I-O"."Drive Lant".WR_AREA,
                  STATUS := "T4 LANT I-O"."Drive Lant".STATUS,
                  "TIME" := "T4 LANT AUX".AUX."TIMER"[18]);
END_REGION

REGION Network 36: T4-LantRost: Referinta Viteza
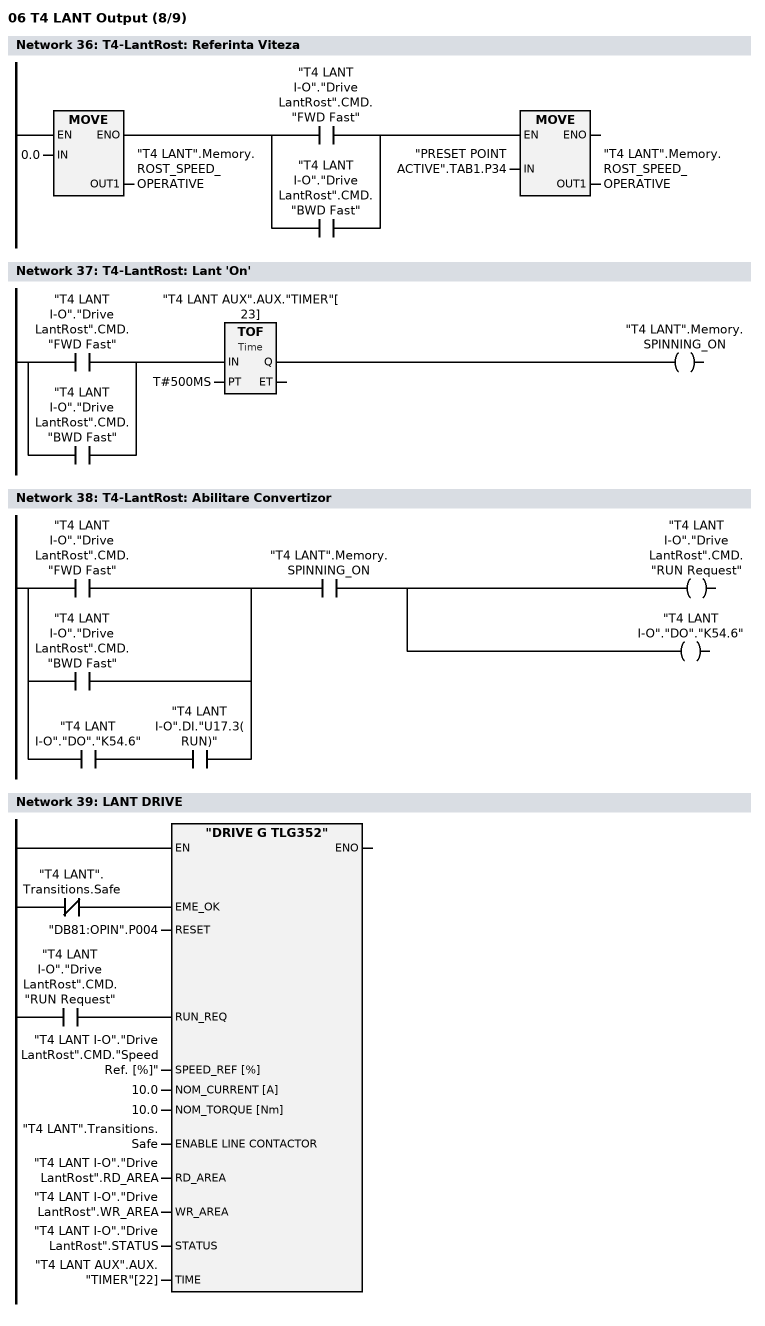
   RUNG wire#powerrail
      Move(in := 0.0, out1 => "T4 LANT".Memory.ROST_SPEED_OPERATIVE)
      wire#w1
      Contact( "T4 LANT I-O"."Drive LantRost".CMD."FWD Fast" )
      wire#w2
      Move(in := "PRESET POINT ACTIVE".TAB1.P34, out1 => "T4 LANT".Memory.ROST_SPEED_OPERATIVE)
   END_RUNG
   RUNG wire#w1
      Contact( "T4 LANT I-O"."Drive LantRost".CMD."BWD Fast" )
   END_RUNG wire#w2
   // the same network as SCL:
   "T4 LANT".Memory.ROST_SPEED_OPERATIVE := 0.0;
   IF "T4 LANT I-O"."Drive LantRost".CMD."FWD Fast" OR "T4 LANT I-O"."Drive LantRost".CMD."BWD Fast" THEN
       "T4 LANT".Memory.ROST_SPEED_OPERATIVE := "PRESET POINT ACTIVE".TAB1.P34;
   END_IF;
END_REGION

REGION Network 37: T4-LantRost: Lant 'On'
   RUNG wire#powerrail
      Contact( "T4 LANT I-O"."Drive LantRost".CMD."FWD Fast" )
      wire#w1
      { S7_Templates := "time_type := Time" } "T4 LANT AUX".AUX."TIMER"[23].TOF(pt := T#500MS, et =>)
      Coil( "T4 LANT".Memory.SPINNING_ON )
   END_RUNG
   RUNG wire#powerrail
      Contact( "T4 LANT I-O"."Drive LantRost".CMD."BWD Fast" )
   END_RUNG wire#w1
   // the same network as SCL:
   "T4 LANT AUX".AUX."TIMER"[23].TOF(IN := "T4 LANT I-O"."Drive LantRost".CMD."FWD Fast" OR "T4 LANT I-O"."Drive LantRost".CMD."BWD Fast",
                           PT := T#500MS);
   "T4 LANT".Memory.SPINNING_ON := "T4 LANT AUX".AUX."TIMER"[23].Q;
END_REGION

REGION Network 38: T4-LantRost: Abilitare Convertizor
   RUNG wire#powerrail
      Contact( "T4 LANT I-O"."Drive LantRost".CMD."FWD Fast" )
      wire#w1
      Contact( "T4 LANT".Memory.SPINNING_ON )
      wire#w2
      Coil( "T4 LANT I-O"."Drive LantRost".CMD."RUN Request" )
   END_RUNG
   RUNG wire#powerrail
      Contact( "T4 LANT I-O"."Drive LantRost".CMD."BWD Fast" )
   END_RUNG wire#w1
   RUNG wire#powerrail
      Contact( "T4 LANT I-O"."DO"."K54.6" )
      Contact( "T4 LANT I-O".DI."U17.3(RUN)" )
   END_RUNG wire#w1
   RUNG wire#w2
      Coil( "T4 LANT I-O"."DO"."K54.6" )
   END_RUNG
   // the same network as SCL:
   "T4 LANT I-O"."Drive LantRost".CMD."RUN Request" := ("T4 LANT I-O"."Drive LantRost".CMD."FWD Fast" OR "T4 LANT I-O"."Drive LantRost".CMD."BWD Fast" OR ("T4 LANT I-O"."DO"."K54.6" AND "T4 LANT I-O".DI."U17.3(RUN)")) AND "T4 LANT".Memory.SPINNING_ON;
   "T4 LANT I-O"."DO"."K54.6" := "T4 LANT I-O"."Drive LantRost".CMD."RUN Request";
END_REGION

REGION Network 39: LANT DRIVE
   RUNG wire#powerrail
      "DRIVE G TLG352"(EME_OK := wire#w1, RUN_REQ := wire#w2, RESET := "DB81:OPIN".P004, "SPEED_REF [%]" := "T4 LANT I-O"."Drive LantRost".CMD."Speed Ref. [%]", "NOM_CURRENT [A]" := 10.0, "NOM_TORQUE [Nm]" := 10.0, "ENABLE LINE CONTACTOR" := "T4 LANT".Transitions.Safe, RD_AREA := "T4 LANT I-O"."Drive LantRost".RD_AREA, WR_AREA := "T4 LANT I-O"."Drive LantRost".WR_AREA, STATUS := "T4 LANT I-O"."Drive LantRost".STATUS, "TIME" := "T4 LANT AUX".AUX."TIMER"[22])
   END_RUNG
   RUNG wire#powerrail
      I_Contact( "T4 LANT".Transitions.Safe )
   END_RUNG wire#w1
   RUNG wire#powerrail
      Contact( "T4 LANT I-O"."Drive LantRost".CMD."RUN Request" )
   END_RUNG wire#w2
   // the same network as SCL:
   "DRIVE G TLG352"(EME_OK := NOT "T4 LANT".Transitions.Safe,
                    RESET := "DB81:OPIN".P004,
                    RUN_REQ := "T4 LANT I-O"."Drive LantRost".CMD."RUN Request",
                    "SPEED_REF [%]" := "T4 LANT I-O"."Drive LantRost".CMD."Speed Ref. [%]",
                    "NOM_CURRENT [A]" := 10.0,
                    "NOM_TORQUE [Nm]" := 10.0,
                    "ENABLE LINE CONTACTOR" := "T4 LANT".Transitions.Safe,
                    RD_AREA := "T4 LANT I-O"."Drive LantRost".RD_AREA,
                    WR_AREA := "T4 LANT I-O"."Drive LantRost".WR_AREA,
                    STATUS := "T4 LANT I-O"."Drive LantRost".STATUS,
                    "TIME" := "T4 LANT AUX".AUX."TIMER"[22]);
END_REGION

REGION Network 40: ================== SEQUENCER STATUS ==================
END_REGION

REGION Network 41: Sequencer Status - Sequence ready to the automatic
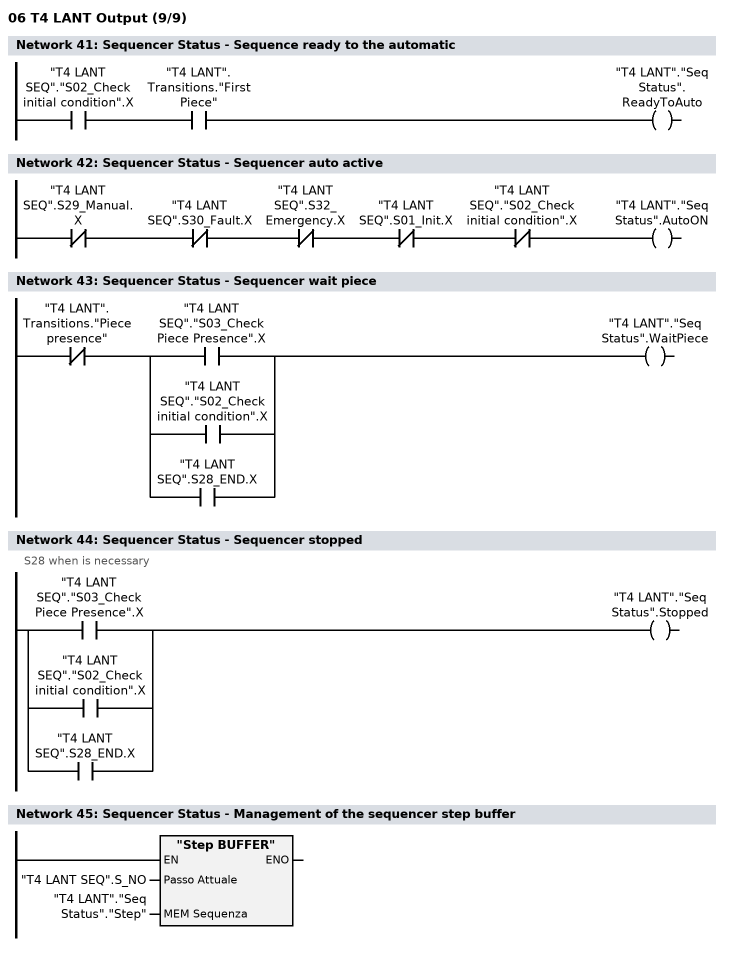
   RUNG wire#powerrail
      Contact( "T4 LANT SEQ"."S02_Check initial condition".X )
      Contact( "T4 LANT".Transitions."First Piece" )
      Coil( "T4 LANT"."Seq Status".ReadyToAuto )
   END_RUNG
   // the same network as SCL:
   "T4 LANT"."Seq Status".ReadyToAuto := "T4 LANT SEQ"."S02_Check initial condition".X AND "T4 LANT".Transitions."First Piece";
END_REGION

REGION Network 42: Sequencer Status - Sequencer auto active
   RUNG wire#powerrail
      I_Contact( "T4 LANT SEQ".S29_Manual.X )
      I_Contact( "T4 LANT SEQ".S30_Fault.X )
      I_Contact( "T4 LANT SEQ".S32_Emergency.X )
      I_Contact( "T4 LANT SEQ".S01_Init.X )
      I_Contact( "T4 LANT SEQ"."S02_Check initial condition".X )
      Coil( "T4 LANT"."Seq Status".AutoON )
   END_RUNG
   // the same network as SCL:
   "T4 LANT"."Seq Status".AutoON := NOT "T4 LANT SEQ".S29_Manual.X AND NOT "T4 LANT SEQ".S30_Fault.X AND NOT "T4 LANT SEQ".S32_Emergency.X AND NOT "T4 LANT SEQ".S01_Init.X AND NOT "T4 LANT SEQ"."S02_Check initial condition".X;
END_REGION

REGION Network 43: Sequencer Status - Sequencer wait piece
   RUNG wire#powerrail
      I_Contact( "T4 LANT".Transitions."Piece presence" )
      wire#w1
      Contact( "T4 LANT SEQ"."S03_Check Piece Presence".X )
      wire#w2
      Coil( "T4 LANT"."Seq Status".WaitPiece )
   END_RUNG
   RUNG wire#w1
      Contact( "T4 LANT SEQ"."S02_Check initial condition".X )
   END_RUNG wire#w2
   RUNG wire#w1
      Contact( "T4 LANT SEQ".S28_END.X )
   END_RUNG wire#w2
   // the same network as SCL:
   "T4 LANT"."Seq Status".WaitPiece := NOT "T4 LANT".Transitions."Piece presence" AND ("T4 LANT SEQ"."S03_Check Piece Presence".X OR "T4 LANT SEQ"."S02_Check initial condition".X OR "T4 LANT SEQ".S28_END.X);
END_REGION

REGION Network 44: Sequencer Status - Sequencer stopped
   // S28 when is necessary
   RUNG wire#powerrail
      Contact( "T4 LANT SEQ"."S03_Check Piece Presence".X )
      wire#w1
      Coil( "T4 LANT"."Seq Status".Stopped )
   END_RUNG
   RUNG wire#powerrail
      Contact( "T4 LANT SEQ"."S02_Check initial condition".X )
   END_RUNG wire#w1
   RUNG wire#powerrail
      Contact( "T4 LANT SEQ".S28_END.X )
   END_RUNG wire#w1
   // the same network as SCL:
   "T4 LANT"."Seq Status".Stopped := "T4 LANT SEQ"."S03_Check Piece Presence".X OR "T4 LANT SEQ"."S02_Check initial condition".X OR "T4 LANT SEQ".S28_END.X;
END_REGION

REGION Network 45: Sequencer Status - Management of the sequencer step buffer
   RUNG wire#powerrail
      "Step BUFFER"("Passo Attuale" := "T4 LANT SEQ".S_NO, "MEM Sequenza" := "T4 LANT"."Seq Status"."Step")
   END_RUNG
   // the same network as SCL:
   "Step BUFFER"("Passo Attuale" := "T4 LANT SEQ".S_NO, "MEM Sequenza" := "T4 LANT"."Seq Status"."Step");
END_REGION
END_FUNCTION
